FUNCTION_BLOCK FB_SaMElementMaintenance EXTENDS FB_SaMElement
VAR
END_VAR

METHOD FB_init : BOOL
VAR_INPUT
	bInitRetains : BOOL; // if TRUE, the retain variables are initialized (warm start / cold start)
	bInCopyCode : BOOL;  // if TRUE, the instance afterwards gets moved into the copy code (online change)
END_VAR
THIS^.SetText (eLocation := E_BaseLocation.pl, wsDescription := "Konserwacja");
THIS^.SetText (eLocation := E_BaseLocation.en, wsDescription := "Maintenance");
THIS^.SetText (eLocation := E_BaseLocation.de, wsDescription := "Wartung");
THIS^.SetName (stName := THIS^.GetTexts ());
END_METHOD

END_FUNCTION_BLOCK

(* stored: Version 1.1.0.1
   POU FB_SaMElementMaintenance: Id {6341cff8-3bbe-0653-0627-63982df4d012}, SpecialFunc None
   Method FB_init: Id {f3bc752e-000f-028b-0a00-bac3729d90de} *)
